TYPE S_SkyCoordEquatorial :
STRUCT
	ra:		LREAL;	// Right Ascension of object  (J2000) in degrees (FK5)
	dec:	LREAL;	// Declination of object (J2000) in degrees (FK5)
END_STRUCT
END_TYPE

(* stored: Version 1.1.0.1, ProductVersion 3.1.4024.12
   DUT S_SkyCoordEquatorial: Id {0bc8efab-a9cb-4bbf-ac60-1625272729f1} *)
